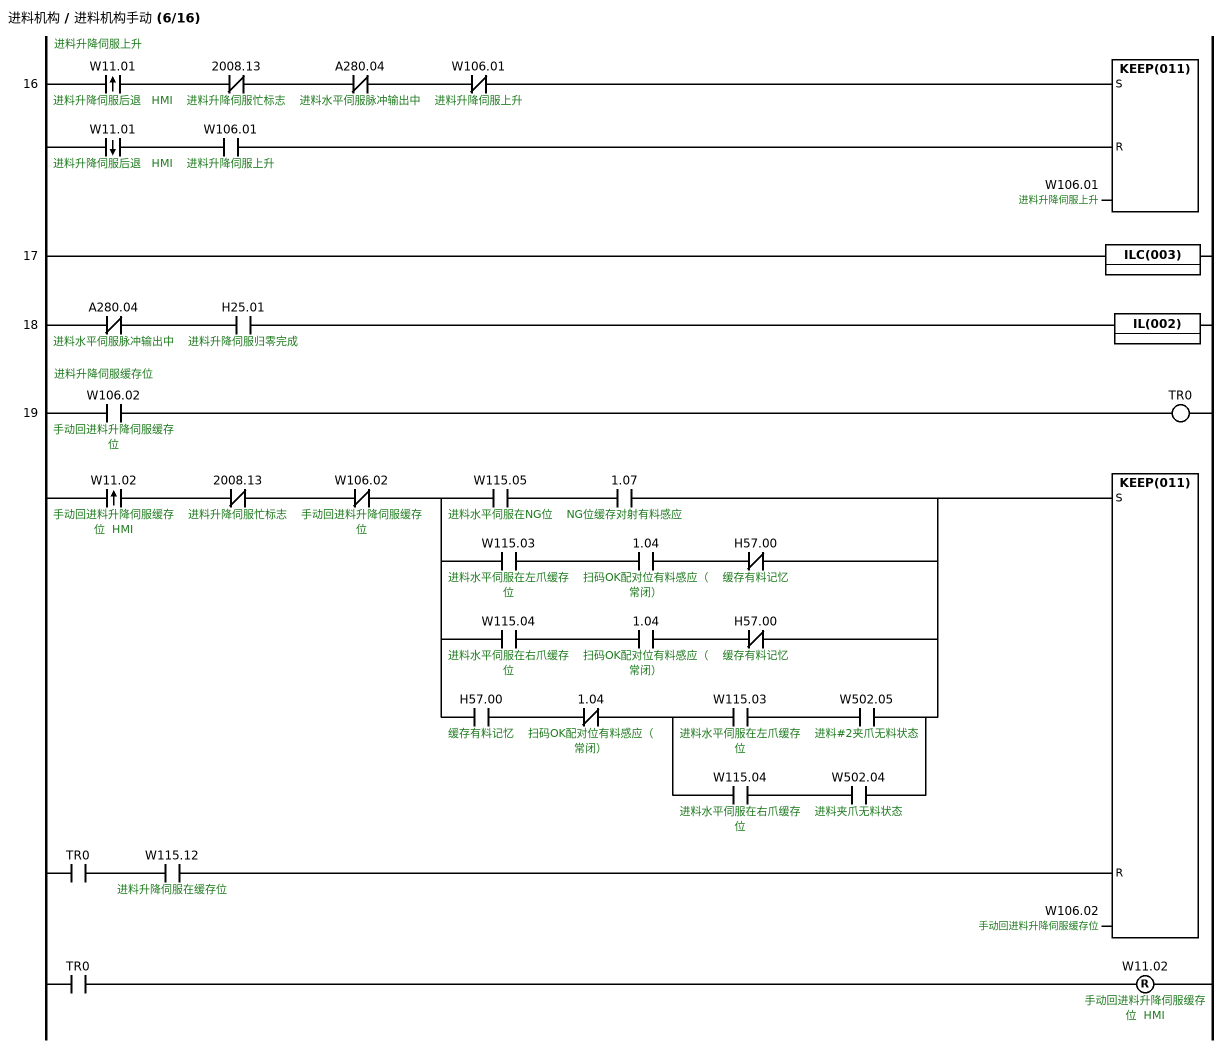
; [picture p120: 进料机构 / 进料机构手动, rungs 16-19]
; rung 16: 进料升降伺服上升
@LD W11.01  ; 进料升降伺服后退   HMI
ANDNOT 2008.13  ; 进料升降伺服忙标志
ANDNOT A280.04  ; 进料水平伺服脉冲输出中
ANDNOT W106.01  ; 进料升降伺服上升
%LD W11.01  ; 进料升降伺服后退   HMI
AND W106.01  ; 进料升降伺服上升
KEEP(011) W106.01  ; 进料升降伺服上升
; rung 17
ILC(003)
; rung 18
LDNOT A280.04  ; 进料水平伺服脉冲输出中
AND H25.01  ; 进料升降伺服归零完成
IL(002)
; rung 19: 进料升降伺服缓存位
@LD W11.02  ; 手动回进料升降伺服缓存位  HMI
ANDNOT 2008.13  ; 进料升降伺服忙标志
ANDNOT W106.02  ; 手动回进料升降伺服缓存位
LD W115.05  ; 进料水平伺服在NG位
AND 1.07  ; NG位缓存对射有料感应
LD W115.03  ; 进料水平伺服在左爪缓存位
AND 1.04  ; 扫码OK配对位有料感应（常闭）
ANDNOT H57.00  ; 缓存有料记忆
ORLD
LD W115.04  ; 进料水平伺服在右爪缓存位
AND 1.04  ; 扫码OK配对位有料感应（常闭）
ANDNOT H57.00  ; 缓存有料记忆
ORLD
LD H57.00  ; 缓存有料记忆
ANDNOT 1.04  ; 扫码OK配对位有料感应（常闭）
LD W115.03  ; 进料水平伺服在左爪缓存位
AND W502.05  ; 进料#2夹爪无料状态
LD W115.04  ; 进料水平伺服在右爪缓存位
AND W502.04  ; 进料夹爪无料状态
ORLD
ANDLD
ORLD
ANDLD
LD W106.02  ; 手动回进料升降伺服缓存位
OUT TR0
AND W115.12  ; 进料升降伺服在缓存位
KEEP(011) W106.02  ; 手动回进料升降伺服缓存位
LD TR0
RSET W11.02  ; 手动回进料升降伺服缓存位  HMI

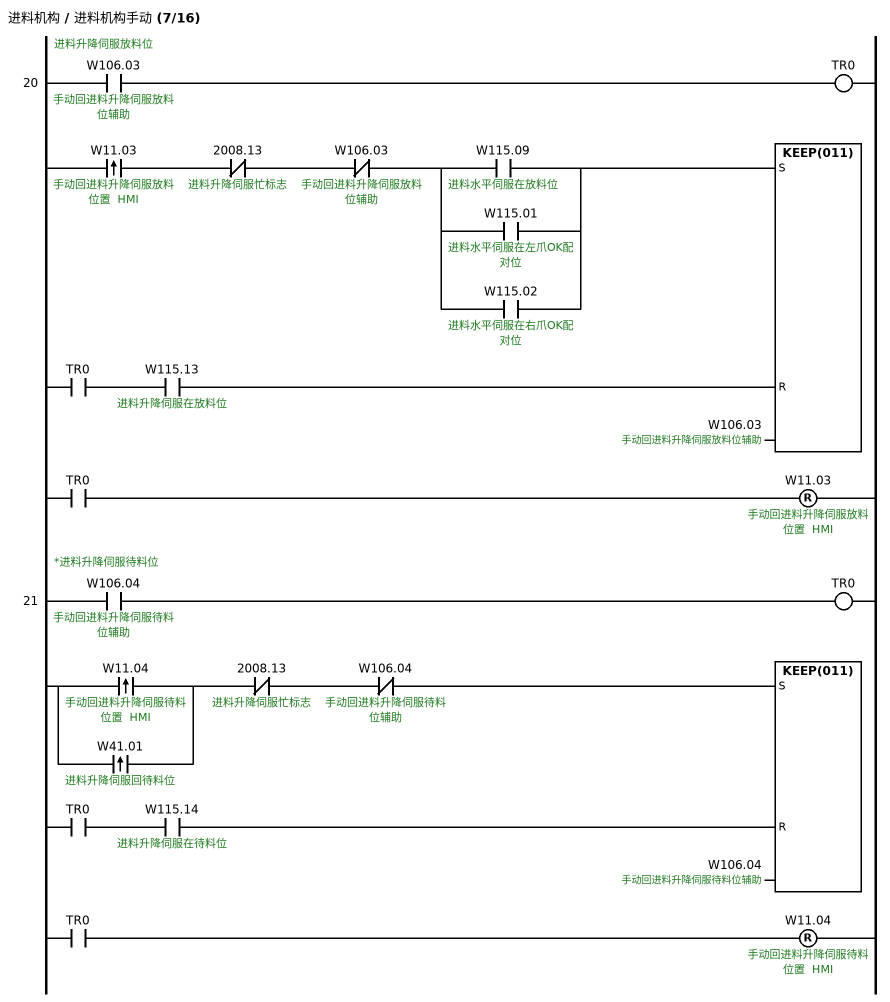
; rung 20: 进料升降伺服放料位
@LD W11.03  ; 手动回进料升降伺服放料位置  HMI
ANDNOT 2008.13  ; 进料升降伺服忙标志
ANDNOT W106.03  ; 手动回进料升降伺服放料位辅助
LD W115.09  ; 进料水平伺服在放料位
OR W115.01  ; 进料水平伺服在左爪OK配对位
OR W115.02  ; 进料水平伺服在右爪OK配对位
ANDLD
LD W106.03  ; 手动回进料升降伺服放料位辅助
OUT TR0
AND W115.13  ; 进料升降伺服在放料位
KEEP(011) W106.03  ; 手动回进料升降伺服放料位辅助
LD TR0
RSET W11.03  ; 手动回进料升降伺服放料位置  HMI
; rung 21: *进料升降伺服待料位
@LD W11.04  ; 手动回进料升降伺服待料位置  HMI
@OR W41.01  ; 进料升降伺服回待料位
ANDNOT 2008.13  ; 进料升降伺服忙标志
ANDNOT W106.04  ; 手动回进料升降伺服待料位辅助
LD W106.04  ; 手动回进料升降伺服待料位辅助
OUT TR0
AND W115.14  ; 进料升降伺服在待料位
KEEP(011) W106.04  ; 手动回进料升降伺服待料位辅助
LD TR0
RSET W11.04  ; 手动回进料升降伺服待料位置  HMI

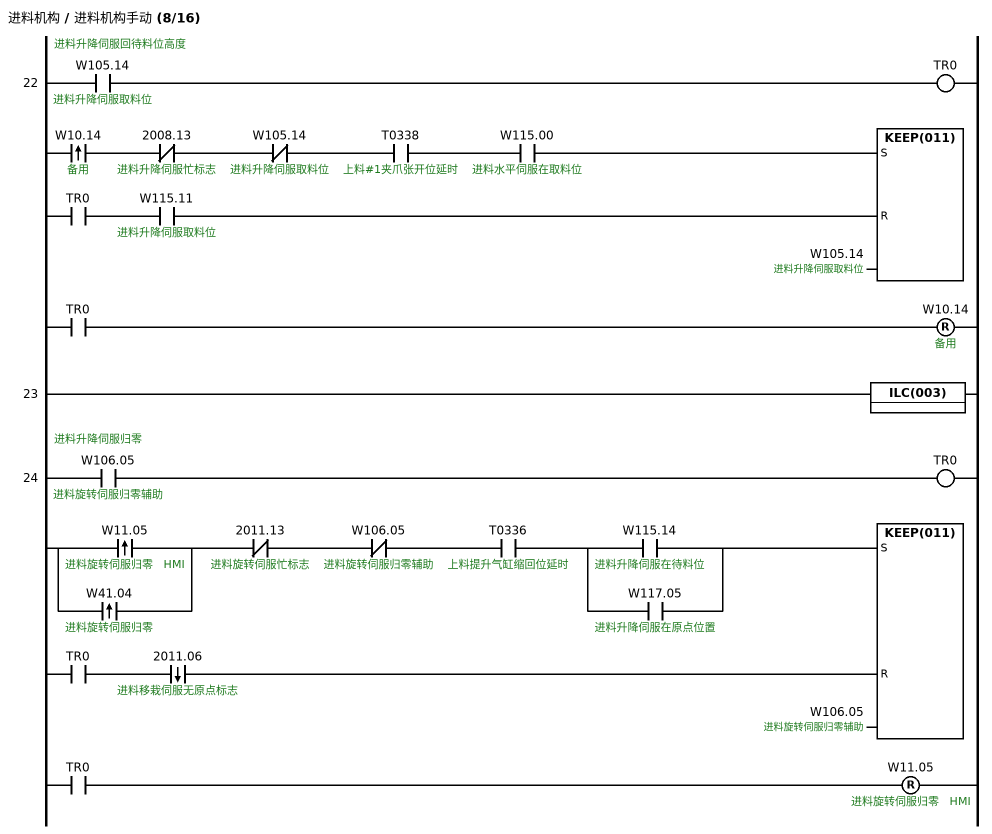
; rung 22: 进料升降伺服回待料位高度
@LD W10.14  ; 备用
ANDNOT 2008.13  ; 进料升降伺服忙标志
ANDNOT W105.14  ; 进料升降伺服取料位
AND T0338  ; 上料#1夹爪张开位延时
AND W115.00  ; 进料水平伺服在取料位
LD W105.14  ; 进料升降伺服取料位
OUT TR0
AND W115.11  ; 进料升降伺服取料位
KEEP(011) W105.14  ; 进料升降伺服取料位
LD TR0
RSET W10.14  ; 备用
; rung 23
ILC(003)
; rung 24: 进料升降伺服归零
@LD W11.05  ; 进料旋转伺服归零   HMI
@OR W41.04  ; 进料旋转伺服归零
ANDNOT 2011.13  ; 进料旋转伺服忙标志
ANDNOT W106.05  ; 进料旋转伺服归零辅助
AND T0336  ; 上料提升气缸缩回位延时
LD W115.14  ; 进料升降伺服在待料位
OR W117.05  ; 进料升降伺服在原点位置
ANDLD
LD W106.05  ; 进料旋转伺服归零辅助
OUT TR0
%AND 2011.06  ; 进料移栽伺服无原点标志
KEEP(011) W106.05  ; 进料旋转伺服归零辅助
LD TR0
RSET W11.05  ; 进料旋转伺服归零   HMI

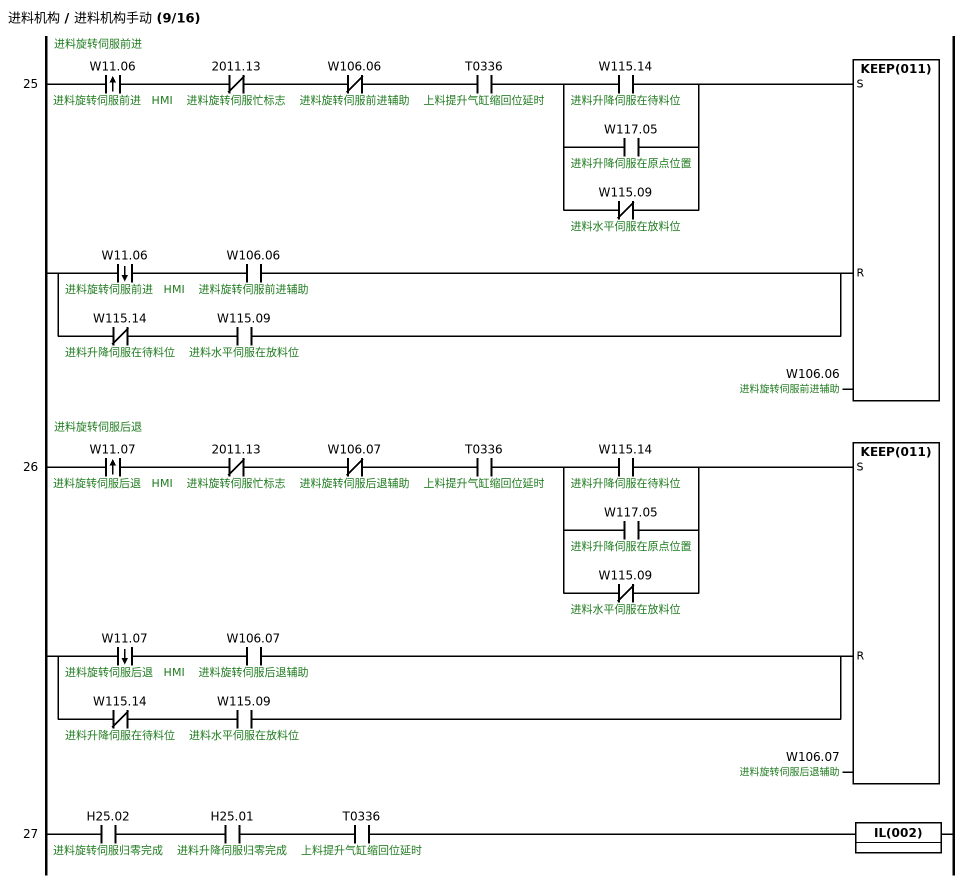
; rung 25: 进料旋转伺服前进
@LD W11.06  ; 进料旋转伺服前进   HMI
ANDNOT 2011.13  ; 进料旋转伺服忙标志
ANDNOT W106.06  ; 进料旋转伺服前进辅助
AND T0336  ; 上料提升气缸缩回位延时
LD W115.14  ; 进料升降伺服在待料位
OR W117.05  ; 进料升降伺服在原点位置
ORNOT W115.09  ; 进料水平伺服在放料位
ANDLD
%LD W11.06  ; 进料旋转伺服前进   HMI
AND W106.06  ; 进料旋转伺服前进辅助
LDNOT W115.14  ; 进料升降伺服在待料位
AND W115.09  ; 进料水平伺服在放料位
ORLD
KEEP(011) W106.06  ; 进料旋转伺服前进辅助
; rung 26: 进料旋转伺服后退
@LD W11.07  ; 进料旋转伺服后退   HMI
ANDNOT 2011.13  ; 进料旋转伺服忙标志
ANDNOT W106.07  ; 进料旋转伺服后退辅助
AND T0336  ; 上料提升气缸缩回位延时
LD W115.14  ; 进料升降伺服在待料位
OR W117.05  ; 进料升降伺服在原点位置
ORNOT W115.09  ; 进料水平伺服在放料位
ANDLD
%LD W11.07  ; 进料旋转伺服后退   HMI
AND W106.07  ; 进料旋转伺服后退辅助
LDNOT W115.14  ; 进料升降伺服在待料位
AND W115.09  ; 进料水平伺服在放料位
ORLD
KEEP(011) W106.07  ; 进料旋转伺服后退辅助
; rung 27
LD H25.02  ; 进料旋转伺服归零完成
AND H25.01  ; 进料升降伺服归零完成
AND T0336  ; 上料提升气缸缩回位延时
IL(002)

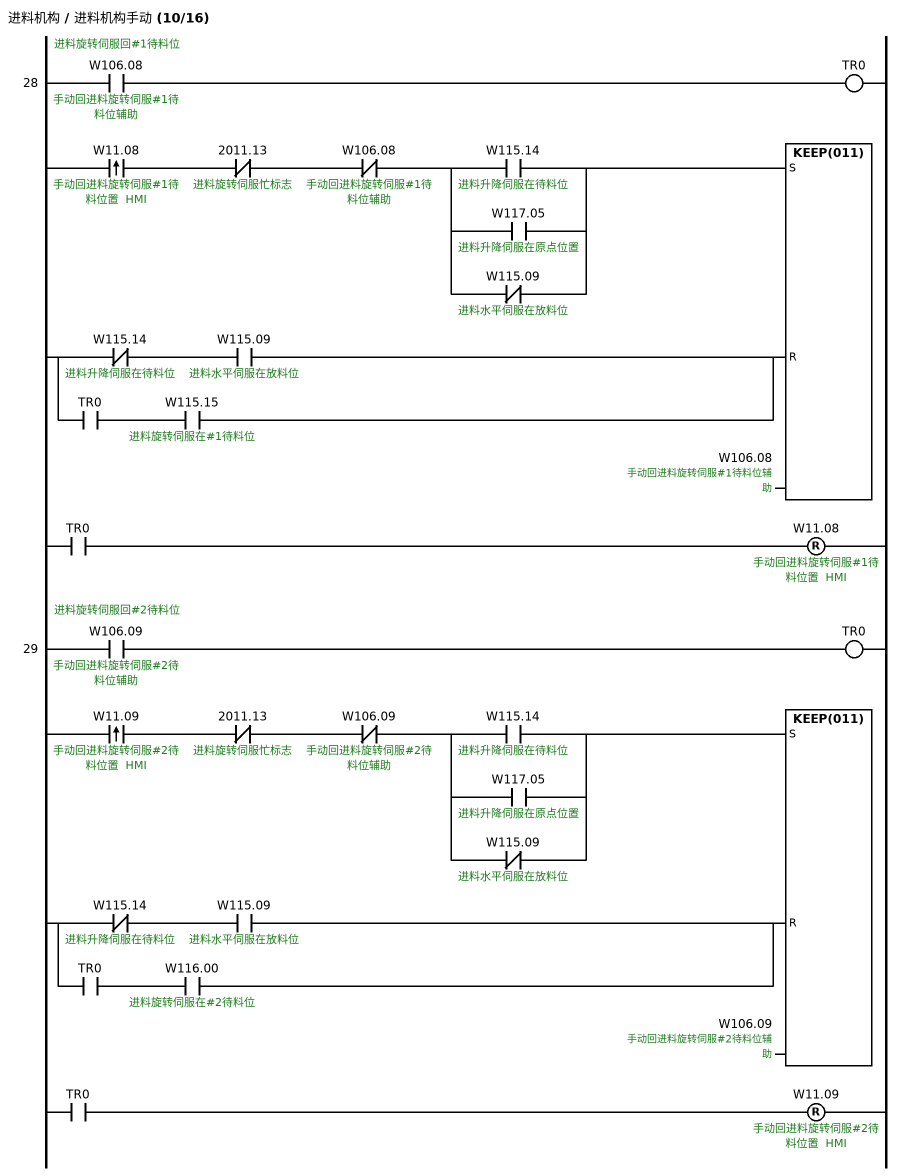
; rung 28: 进料旋转伺服回#1待料位
@LD W11.08  ; 手动回进料旋转伺服#1待料位置  HMI
ANDNOT 2011.13  ; 进料旋转伺服忙标志
ANDNOT W106.08  ; 手动回进料旋转伺服#1待料位辅助
LD W115.14  ; 进料升降伺服在待料位
OR W117.05  ; 进料升降伺服在原点位置
ORNOT W115.09  ; 进料水平伺服在放料位
ANDLD
LDNOT W115.14  ; 进料升降伺服在待料位
AND W115.09  ; 进料水平伺服在放料位
LD W106.08  ; 手动回进料旋转伺服#1待料位辅助
OUT TR0
AND W115.15  ; 进料旋转伺服在#1待料位
ORLD
KEEP(011) W106.08  ; 手动回进料旋转伺服#1待料位辅助
LD TR0
RSET W11.08  ; 手动回进料旋转伺服#1待料位置  HMI
; rung 29: 进料旋转伺服回#2待料位
@LD W11.09  ; 手动回进料旋转伺服#2待料位置  HMI
ANDNOT 2011.13  ; 进料旋转伺服忙标志
ANDNOT W106.09  ; 手动回进料旋转伺服#2待料位辅助
LD W115.14  ; 进料升降伺服在待料位
OR W117.05  ; 进料升降伺服在原点位置
ORNOT W115.09  ; 进料水平伺服在放料位
ANDLD
LDNOT W115.14  ; 进料升降伺服在待料位
AND W115.09  ; 进料水平伺服在放料位
LD W106.09  ; 手动回进料旋转伺服#2待料位辅助
OUT TR0
AND W116.00  ; 进料旋转伺服在#2待料位
ORLD
KEEP(011) W106.09  ; 手动回进料旋转伺服#2待料位辅助
LD TR0
RSET W11.09  ; 手动回进料旋转伺服#2待料位置  HMI

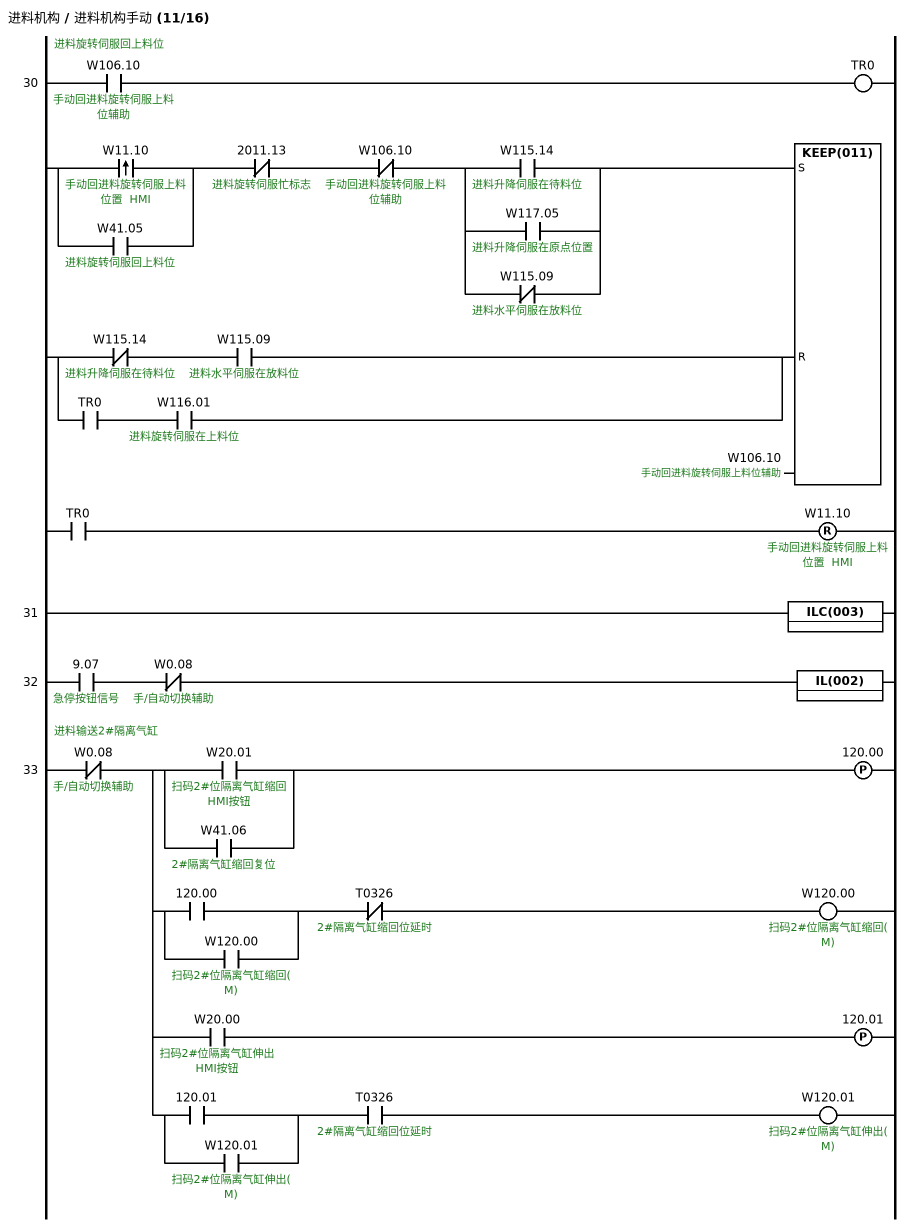
; rung 30: 进料旋转伺服回上料位
@LD W11.10  ; 手动回进料旋转伺服上料位置  HMI
OR W41.05  ; 进料旋转伺服回上料位
ANDNOT 2011.13  ; 进料旋转伺服忙标志
ANDNOT W106.10  ; 手动回进料旋转伺服上料位辅助
LD W115.14  ; 进料升降伺服在待料位
OR W117.05  ; 进料升降伺服在原点位置
ORNOT W115.09  ; 进料水平伺服在放料位
ANDLD
LDNOT W115.14  ; 进料升降伺服在待料位
AND W115.09  ; 进料水平伺服在放料位
LD W106.10  ; 手动回进料旋转伺服上料位辅助
OUT TR0
AND W116.01  ; 进料旋转伺服在上料位
ORLD
KEEP(011) W106.10  ; 手动回进料旋转伺服上料位辅助
LD TR0
RSET W11.10  ; 手动回进料旋转伺服上料位置  HMI
; rung 31
ILC(003)
; rung 32
LD 9.07  ; 急停按钮信号
ANDNOT W0.08  ; 手/自动切换辅助
IL(002)
; rung 33: 进料输送2#隔离气缸
LDNOT W0.08  ; 手/自动切换辅助
OUT TR0
LD W20.01  ; 扫码2#位隔离气缸缩回   HMI按钮
OR W41.06  ; 2#隔离气缸缩回复位
ANDLD
DIFU(013) 120.00
LD TR0
LD 120.00
OR W120.00  ; 扫码2#位隔离气缸缩回(M)
ANDLD
ANDNOT T0326  ; 2#隔离气缸缩回位延时
OUT W120.00  ; 扫码2#位隔离气缸缩回(M)
LD TR0
AND W20.00  ; 扫码2#位隔离气缸伸出   HMI按钮
DIFU(013) 120.01
LD TR0
LD 120.01
OR W120.01  ; 扫码2#位隔离气缸伸出(M)
ANDLD
AND T0326  ; 2#隔离气缸缩回位延时
OUT W120.01  ; 扫码2#位隔离气缸伸出(M)

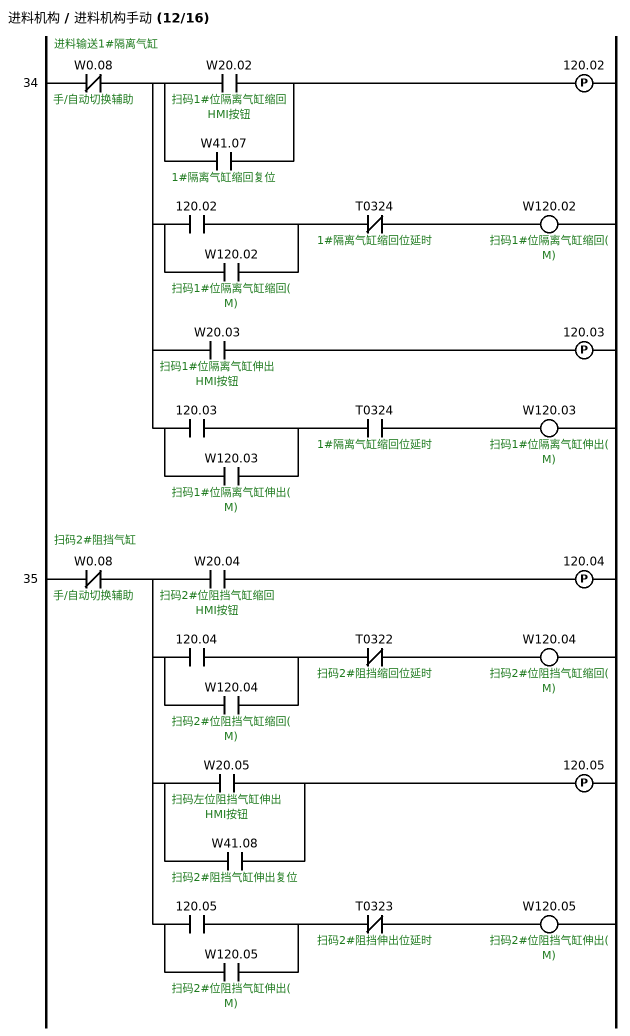
; rung 34: 进料输送1#隔离气缸
LDNOT W0.08  ; 手/自动切换辅助
OUT TR0
LD W20.02  ; 扫码1#位隔离气缸缩回   HMI按钮
OR W41.07  ; 1#隔离气缸缩回复位
ANDLD
DIFU(013) 120.02
LD TR0
LD 120.02
OR W120.02  ; 扫码1#位隔离气缸缩回(M)
ANDLD
ANDNOT T0324  ; 1#隔离气缸缩回位延时
OUT W120.02  ; 扫码1#位隔离气缸缩回(M)
LD TR0
AND W20.03  ; 扫码1#位隔离气缸伸出   HMI按钮
DIFU(013) 120.03
LD TR0
LD 120.03
OR W120.03  ; 扫码1#位隔离气缸伸出(M)
ANDLD
AND T0324  ; 1#隔离气缸缩回位延时
OUT W120.03  ; 扫码1#位隔离气缸伸出(M)
; rung 35: 扫码2#阻挡气缸
LDNOT W0.08  ; 手/自动切换辅助
OUT TR0
AND W20.04  ; 扫码2#位阻挡气缸缩回   HMI按钮
DIFU(013) 120.04
LD TR0
LD 120.04
OR W120.04  ; 扫码2#位阻挡气缸缩回(M)
ANDLD
ANDNOT T0322  ; 扫码2#阻挡缩回位延时
OUT W120.04  ; 扫码2#位阻挡气缸缩回(M)
LD TR0
LD W20.05  ; 扫码左位阻挡气缸伸出  HMI按钮
OR W41.08  ; 扫码2#阻挡气缸伸出复位
ANDLD
DIFU(013) 120.05
LD TR0
LD 120.05
OR W120.05  ; 扫码2#位阻挡气缸伸出(M)
ANDLD
ANDNOT T0323  ; 扫码2#阻挡伸出位延时
OUT W120.05  ; 扫码2#位阻挡气缸伸出(M)

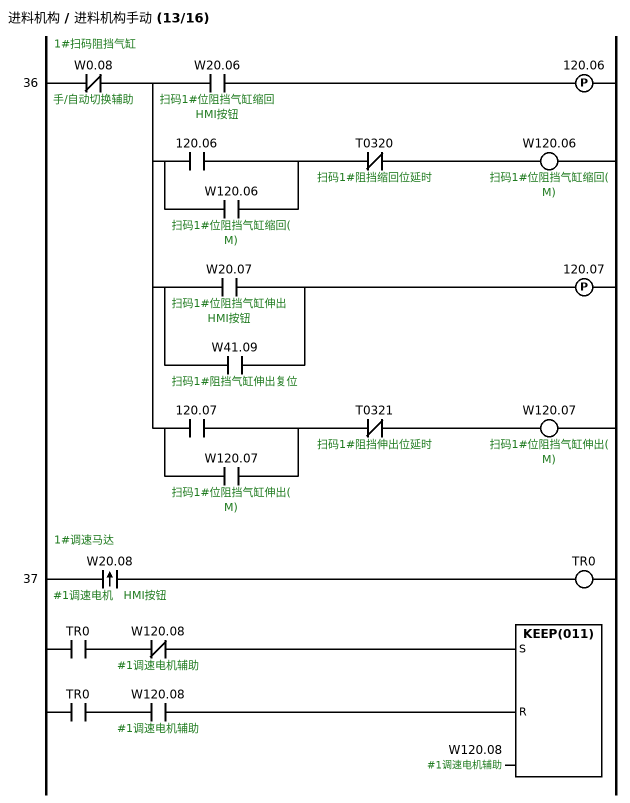
; rung 36: 1#扫码阻挡气缸
LDNOT W0.08  ; 手/自动切换辅助
OUT TR0
AND W20.06  ; 扫码1#位阻挡气缸缩回   HMI按钮
DIFU(013) 120.06
LD TR0
LD 120.06
OR W120.06  ; 扫码1#位阻挡气缸缩回(M)
ANDLD
ANDNOT T0320  ; 扫码1#阻挡缩回位延时
OUT W120.06  ; 扫码1#位阻挡气缸缩回(M)
LD TR0
LD W20.07  ; 扫码1#位阻挡气缸伸出   HMI按钮
OR W41.09  ; 扫码1#阻挡气缸伸出复位
ANDLD
DIFU(013) 120.07
LD TR0
LD 120.07
OR W120.07  ; 扫码1#位阻挡气缸伸出(M)
ANDLD
ANDNOT T0321  ; 扫码1#阻挡伸出位延时
OUT W120.07  ; 扫码1#位阻挡气缸伸出(M)
; rung 37: 1#调速马达
@LD W20.08  ; #1调速电机   HMI按钮
OUT TR0
ANDNOT W120.08  ; #1调速电机辅助
LD TR0
AND W120.08  ; #1调速电机辅助
KEEP(011) W120.08  ; #1调速电机辅助

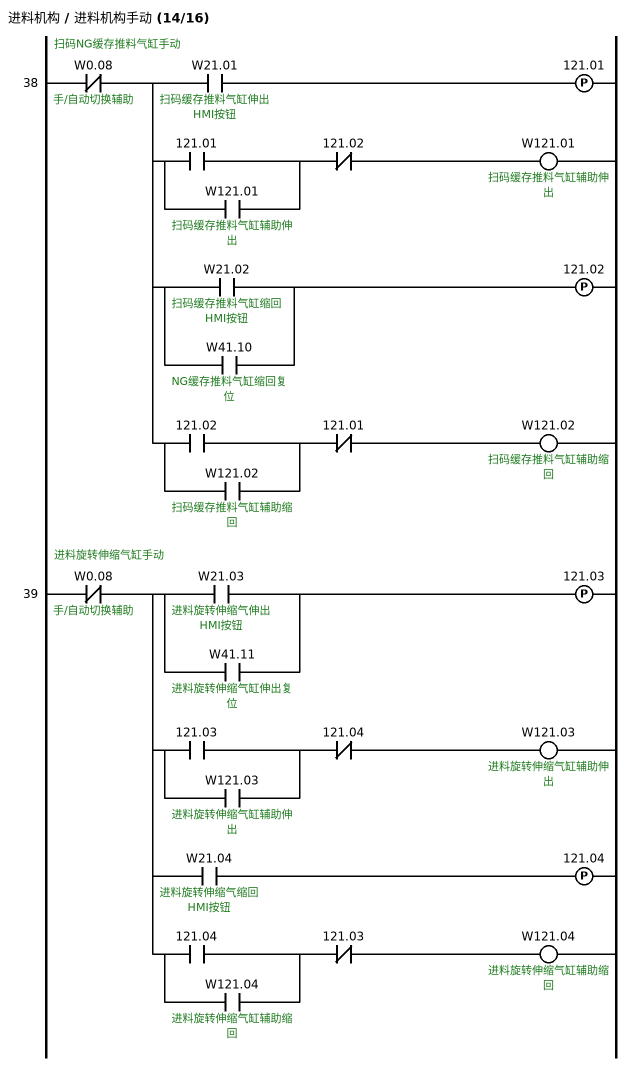
; rung 38: 扫码NG缓存推料气缸手动
LDNOT W0.08  ; 手/自动切换辅助
OUT TR0
AND W21.01  ; 扫码缓存推料气缸伸出   HMI按钮
DIFU(013) 121.01
LD TR0
LD 121.01
OR W121.01  ; 扫码缓存推料气缸辅助伸出
ANDLD
ANDNOT 121.02
OUT W121.01  ; 扫码缓存推料气缸辅助伸出
LD TR0
LD W21.02  ; 扫码缓存推料气缸缩回   HMI按钮
OR W41.10  ; NG缓存推料气缸缩回复位
ANDLD
DIFU(013) 121.02
LD TR0
LD 121.02
OR W121.02  ; 扫码缓存推料气缸辅助缩回
ANDLD
ANDNOT 121.01
OUT W121.02  ; 扫码缓存推料气缸辅助缩回
; rung 39: 进料旋转伸缩气缸手动
LDNOT W0.08  ; 手/自动切换辅助
OUT TR0
LD W21.03  ; 进料旋转伸缩气伸出   HMI按钮
OR W41.11  ; 进料旋转伸缩气缸伸出复位
ANDLD
DIFU(013) 121.03
LD TR0
LD 121.03
OR W121.03  ; 进料旋转伸缩气缸辅助伸出
ANDLD
ANDNOT 121.04
OUT W121.03  ; 进料旋转伸缩气缸辅助伸出
LD TR0
AND W21.04  ; 进料旋转伸缩气缩回   HMI按钮
DIFU(013) 121.04
LD TR0
LD 121.04
OR W121.04  ; 进料旋转伸缩气缸辅助缩回
ANDLD
ANDNOT 121.03
OUT W121.04  ; 进料旋转伸缩气缸辅助缩回

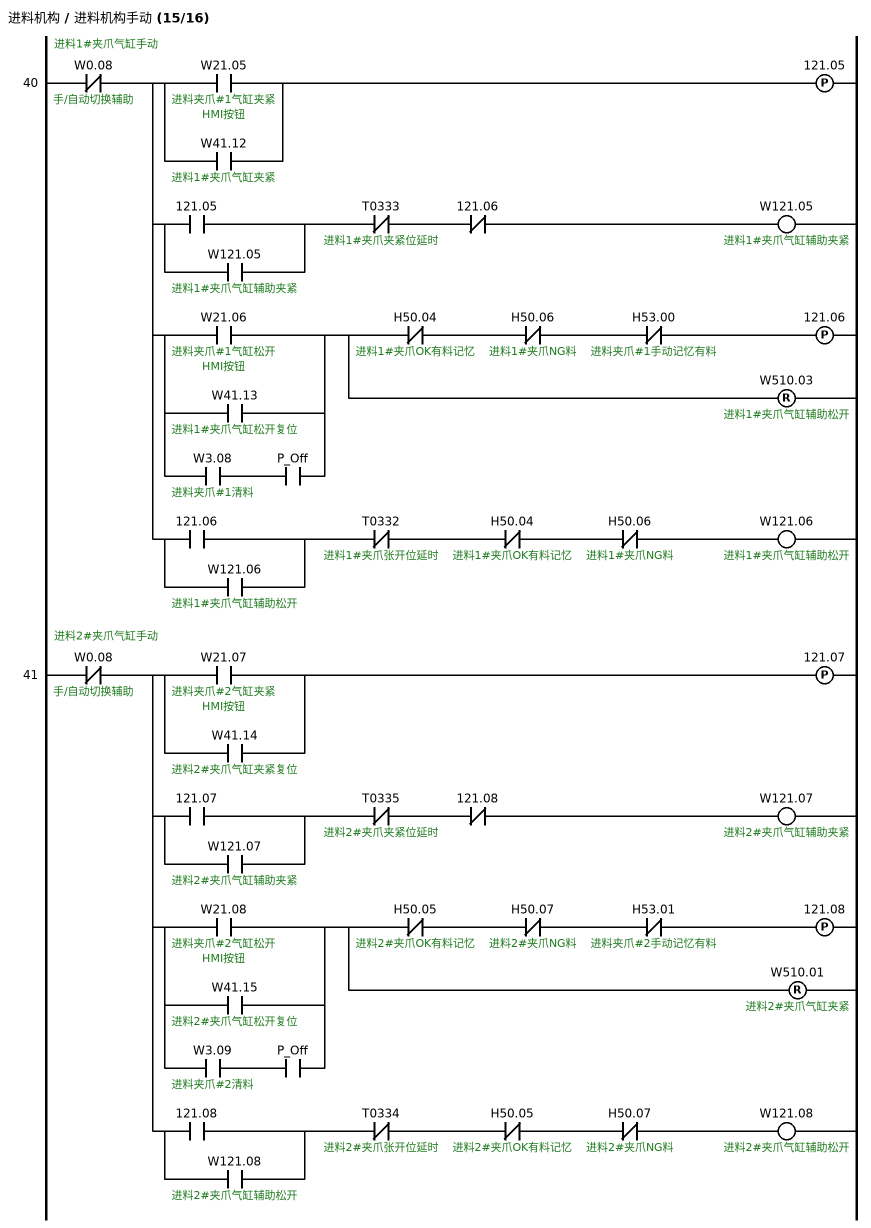
; rung 40: 进料1#夹爪气缸手动
LDNOT W0.08  ; 手/自动切换辅助
OUT TR0
LD W21.05  ; 进料夹爪#1气缸夹紧   HMI按钮
OR W41.12  ; 进料1#夹爪气缸夹紧
ANDLD
DIFU(013) 121.05
LD TR0
LD 121.05
OR W121.05  ; 进料1#夹爪气缸辅助夹紧
ANDLD
ANDNOT T0333  ; 进料1#夹爪夹紧位延时
ANDNOT 121.06
OUT W121.05  ; 进料1#夹爪气缸辅助夹紧
LD TR0
LD W21.06  ; 进料夹爪#1气缸松开   HMI按钮
OR W41.13  ; 进料1#夹爪气缸松开复位
LD W3.08  ; 进料夹爪#1清料
AND P_Off
ORLD
ANDLD
OUT TR1
ANDNOT H50.04  ; 进料1#夹爪OK有料记忆
ANDNOT H50.06  ; 进料1#夹爪NG料
ANDNOT H53.00  ; 进料夹爪#1手动记忆有料
DIFU(013) 121.06
LD TR1
RSET W510.03  ; 进料1#夹爪气缸辅助松开
LD TR0
LD 121.06
OR W121.06  ; 进料1#夹爪气缸辅助松开
ANDLD
ANDNOT T0332  ; 进料1#夹爪张开位延时
ANDNOT H50.04  ; 进料1#夹爪OK有料记忆
ANDNOT H50.06  ; 进料1#夹爪NG料
OUT W121.06  ; 进料1#夹爪气缸辅助松开
; rung 41: 进料2#夹爪气缸手动
LDNOT W0.08  ; 手/自动切换辅助
OUT TR0
LD W21.07  ; 进料夹爪#2气缸夹紧   HMI按钮
OR W41.14  ; 进料2#夹爪气缸夹紧复位
ANDLD
DIFU(013) 121.07
LD TR0
LD 121.07
OR W121.07  ; 进料2#夹爪气缸辅助夹紧
ANDLD
ANDNOT T0335  ; 进料2#夹爪夹紧位延时
ANDNOT 121.08
OUT W121.07  ; 进料2#夹爪气缸辅助夹紧
LD TR0
LD W21.08  ; 进料夹爪#2气缸松开   HMI按钮
OR W41.15  ; 进料2#夹爪气缸松开复位
LD W3.09  ; 进料夹爪#2清料
AND P_Off
ORLD
ANDLD
OUT TR1
ANDNOT H50.05  ; 进料2#夹爪OK有料记忆
ANDNOT H50.07  ; 进料2#夹爪NG料
ANDNOT H53.01  ; 进料夹爪#2手动记忆有料
DIFU(013) 121.08
LD TR1
RSET W510.01  ; 进料2#夹爪气缸夹紧
LD TR0
LD 121.08
OR W121.08  ; 进料2#夹爪气缸辅助松开
ANDLD
ANDNOT T0334  ; 进料2#夹爪张开位延时
ANDNOT H50.05  ; 进料2#夹爪OK有料记忆
ANDNOT H50.07  ; 进料2#夹爪NG料
OUT W121.08  ; 进料2#夹爪气缸辅助松开

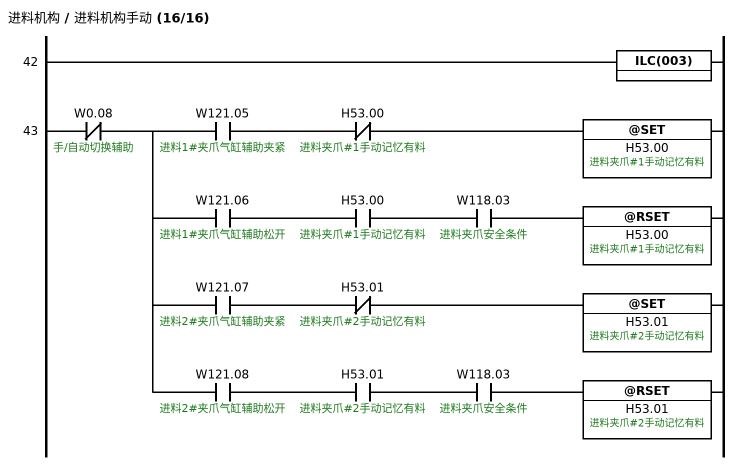
; rung 42
ILC(003)
; rung 43
LDNOT W0.08  ; 手/自动切换辅助
OUT TR0
AND W121.05  ; 进料1#夹爪气缸辅助夹紧
ANDNOT H53.00  ; 进料夹爪#1手动记忆有料
@SET H53.00  ; 进料夹爪#1手动记忆有料
LD TR0
AND W121.06  ; 进料1#夹爪气缸辅助松开
AND H53.00  ; 进料夹爪#1手动记忆有料
AND W118.03  ; 进料夹爪安全条件
@RSET H53.00  ; 进料夹爪#1手动记忆有料
LD TR0
AND W121.07  ; 进料2#夹爪气缸辅助夹紧
ANDNOT H53.01  ; 进料夹爪#2手动记忆有料
@SET H53.01  ; 进料夹爪#2手动记忆有料
LD TR0
AND W121.08  ; 进料2#夹爪气缸辅助松开
AND H53.01  ; 进料夹爪#2手动记忆有料
AND W118.03  ; 进料夹爪安全条件
@RSET H53.01  ; 进料夹爪#2手动记忆有料

### Section 进料水平伺服参数设置

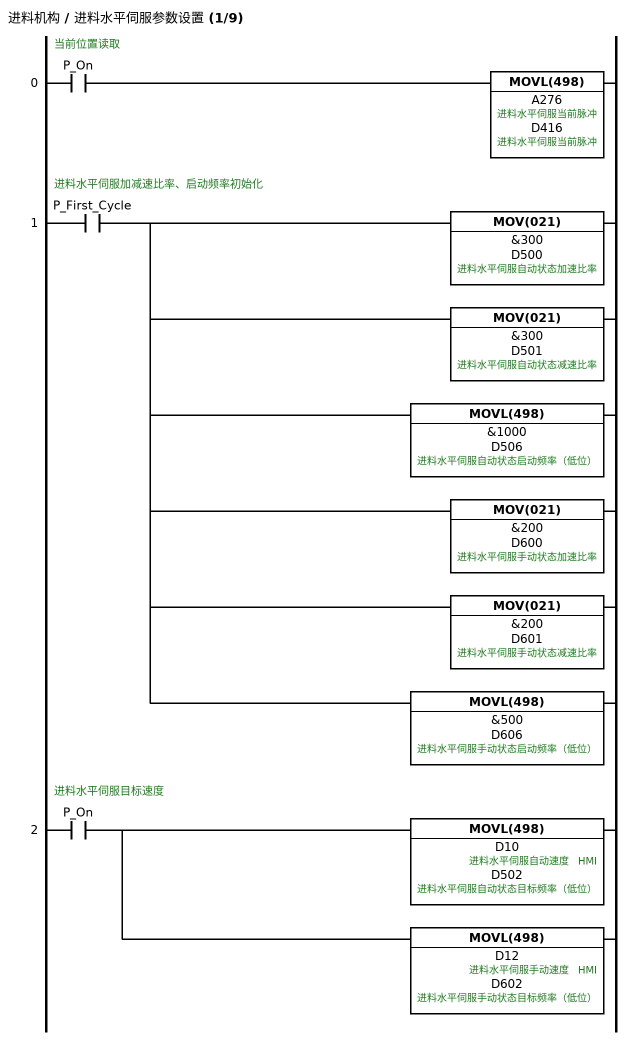
; rung 0: 当前位置读取
LD P_On
MOVL(498) A276 D416  ; 进料水平伺服当前脉冲
; rung 1: 进料水平伺服加减速比率、启动频率初始化
LD P_First_Cycle
MOV(021) &300 D500  ; 进料水平伺服自动状态加速比率
MOV(021) &300 D501  ; 进料水平伺服自动状态减速比率
MOVL(498) &1000 D506  ; 进料水平伺服自动状态启动频率（低位）
MOV(021) &200 D600  ; 进料水平伺服手动状态加速比率
MOV(021) &200 D601  ; 进料水平伺服手动状态减速比率
MOVL(498) &500 D606  ; 进料水平伺服手动状态启动频率（低位）
; rung 2: 进料水平伺服目标速度
LD P_On
MOVL(498) D10 D502  ; 进料水平伺服自动速度   HMI, 进料水平伺服自动状态目标频率（低位）
MOVL(498) D12 D602  ; 进料水平伺服手动速度   HMI, 进料水平伺服手动状态目标频率（低位）

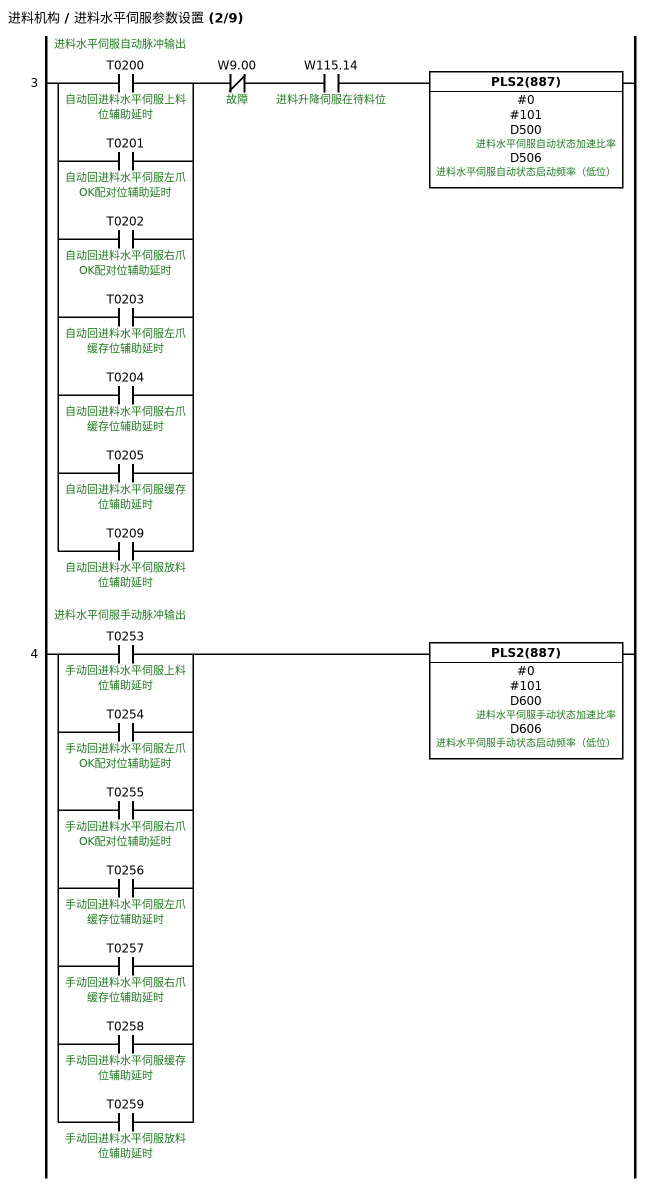
; rung 3: 进料水平伺服自动脉冲输出
LD T0200  ; 自动回进料水平伺服上料位辅助延时
OR T0201  ; 自动回进料水平伺服左爪OK配对位辅助延时
OR T0202  ; 自动回进料水平伺服右爪OK配对位辅助延时
OR T0203  ; 自动回进料水平伺服左爪缓存位辅助延时
OR T0204  ; 自动回进料水平伺服右爪缓存位辅助延时
OR T0205  ; 自动回进料水平伺服缓存位辅助延时
OR T0209  ; 自动回进料水平伺服放料位辅助延时
ANDNOT W9.00  ; 故障
AND W115.14  ; 进料升降伺服在待料位
PLS2(887) #0 #101 D500 D506  ; 进料水平伺服自动状态加速比率, 进料水平伺服自动状态启动频率（低位）
; rung 4: 进料水平伺服手动脉冲输出
LD T0253  ; 手动回进料水平伺服上料位辅助延时
OR T0254  ; 手动回进料水平伺服左爪OK配对位辅助延时
OR T0255  ; 手动回进料水平伺服右爪OK配对位辅助延时
OR T0256  ; 手动回进料水平伺服左爪缓存位辅助延时
OR T0257  ; 手动回进料水平伺服右爪缓存位辅助延时
OR T0258  ; 手动回进料水平伺服缓存位辅助延时
OR T0259  ; 手动回进料水平伺服放料位辅助延时
PLS2(887) #0 #101 D600 D606  ; 进料水平伺服手动状态加速比率, 进料水平伺服手动状态启动频率（低位）

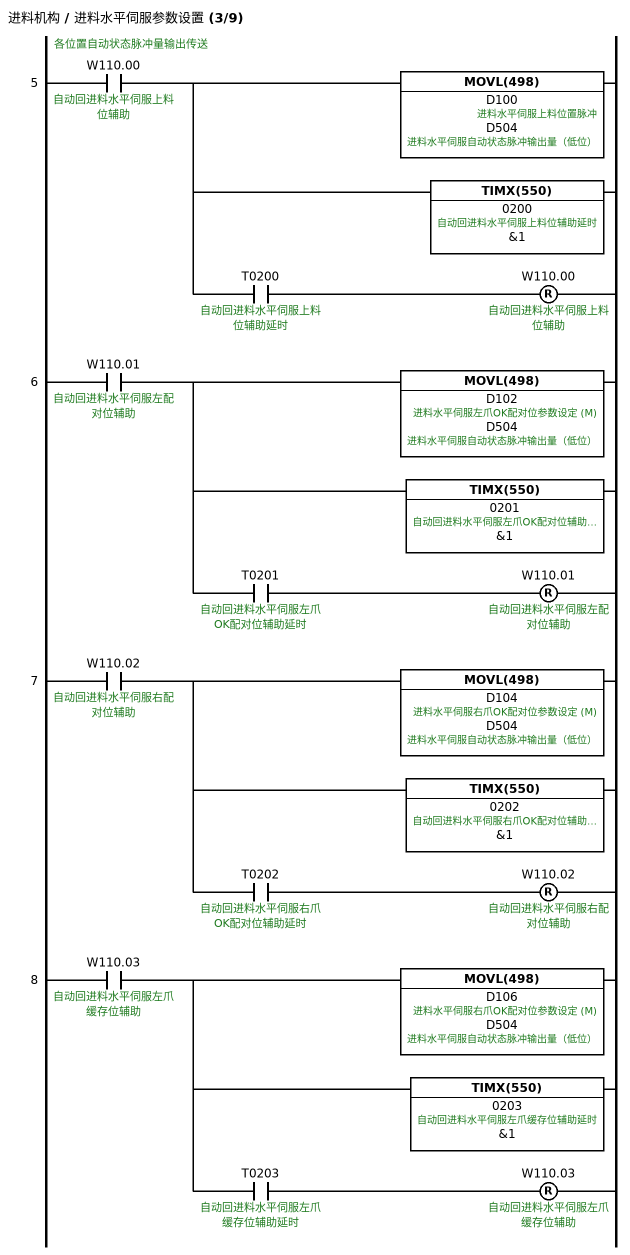
; rung 5: 各位置自动状态脉冲量输出传送
LD W110.00  ; 自动回进料水平伺服上料位辅助
MOVL(498) D100 D504  ; 进料水平伺服上料位置脉冲, 进料水平伺服自动状态脉冲输出量（低位）
TIMX(550) 0200 &1  ; 自动回进料水平伺服上料位辅助延时
AND T0200  ; 自动回进料水平伺服上料位辅助延时
RSET W110.00  ; 自动回进料水平伺服上料位辅助
; rung 6
LD W110.01  ; 自动回进料水平伺服左配对位辅助
MOVL(498) D102 D504  ; 进料水平伺服左爪OK配对位参数设定 (M), 进料水平伺服自动状态脉冲输出量（低位）
TIMX(550) 0201 &1  ; 自动回进料水平伺服左爪OK配对位辅助延时
AND T0201  ; 自动回进料水平伺服左爪OK配对位辅助延时
RSET W110.01  ; 自动回进料水平伺服左配对位辅助
; rung 7
LD W110.02  ; 自动回进料水平伺服右配对位辅助
MOVL(498) D104 D504  ; 进料水平伺服右爪OK配对位参数设定 (M), 进料水平伺服自动状态脉冲输出量（低位）
TIMX(550) 0202 &1  ; 自动回进料水平伺服右爪OK配对位辅助延时
AND T0202  ; 自动回进料水平伺服右爪OK配对位辅助延时
RSET W110.02  ; 自动回进料水平伺服右配对位辅助
; rung 8
LD W110.03  ; 自动回进料水平伺服左爪缓存位辅助
MOVL(498) D106 D504  ; 进料水平伺服右爪OK配对位参数设定 (M), 进料水平伺服自动状态脉冲输出量（低位）
TIMX(550) 0203 &1  ; 自动回进料水平伺服左爪缓存位辅助延时
AND T0203  ; 自动回进料水平伺服左爪缓存位辅助延时
RSET W110.03  ; 自动回进料水平伺服左爪缓存位辅助

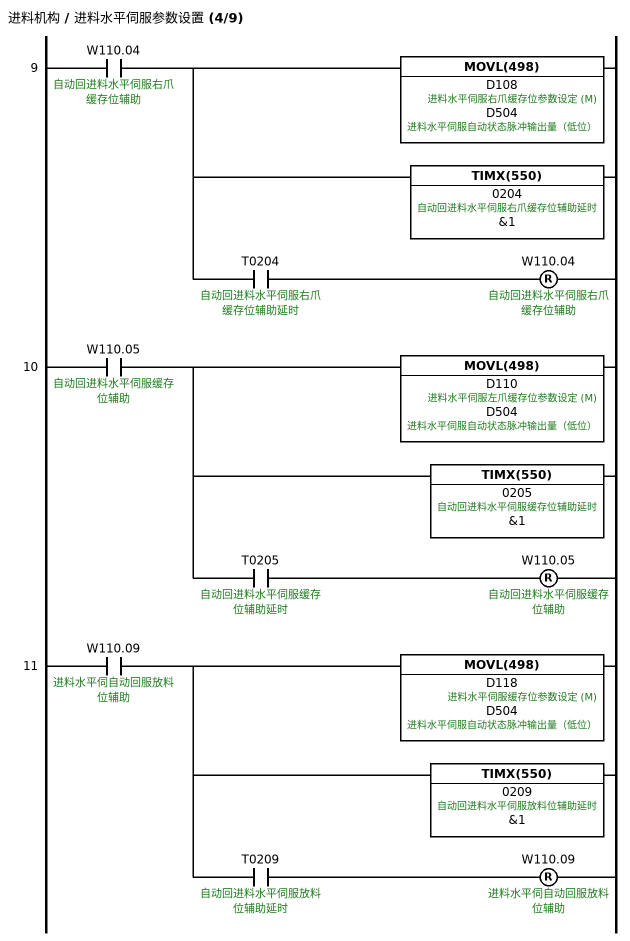
; rung 9
LD W110.04  ; 自动回进料水平伺服右爪缓存位辅助
MOVL(498) D108 D504  ; 进料水平伺服右爪缓存位参数设定 (M), 进料水平伺服自动状态脉冲输出量（低位）
TIMX(550) 0204 &1  ; 自动回进料水平伺服右爪缓存位辅助延时
AND T0204  ; 自动回进料水平伺服右爪缓存位辅助延时
RSET W110.04  ; 自动回进料水平伺服右爪缓存位辅助
; rung 10
LD W110.05  ; 自动回进料水平伺服缓存位辅助
MOVL(498) D110 D504  ; 进料水平伺服左爪缓存位参数设定 (M), 进料水平伺服自动状态脉冲输出量（低位）
TIMX(550) 0205 &1  ; 自动回进料水平伺服缓存位辅助延时
AND T0205  ; 自动回进料水平伺服缓存位辅助延时
RSET W110.05  ; 自动回进料水平伺服缓存位辅助
; rung 11
LD W110.09  ; 进料水平伺自动回服放料位辅助
MOVL(498) D118 D504  ; 进料水平伺服缓存位参数设定 (M), 进料水平伺服自动状态脉冲输出量（低位）
TIMX(550) 0209 &1  ; 自动回进料水平伺服放料位辅助延时
AND T0209  ; 自动回进料水平伺服放料位辅助延时
RSET W110.09  ; 进料水平伺自动回服放料位辅助

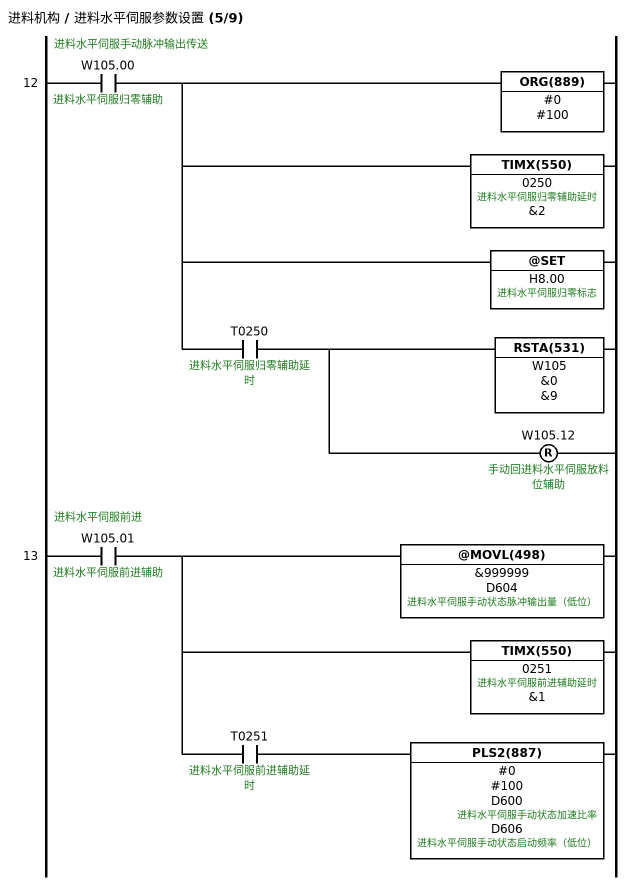
; rung 12: 进料水平伺服手动脉冲输出传送
LD W105.00  ; 进料水平伺服归零辅助
ORG(889) #0 #100
TIMX(550) 0250 &2  ; 进料水平伺服归零辅助延时
@SET H8.00  ; 进料水平伺服归零标志
AND T0250  ; 进料水平伺服归零辅助延时
RSTA(531) W105 &0 &9
RSET W105.12  ; 手动回进料水平伺服放料位辅助
; rung 13: 进料水平伺服前进
LD W105.01  ; 进料水平伺服前进辅助
@MOVL(498) &999999 D604  ; 进料水平伺服手动状态脉冲输出量（低位）
TIMX(550) 0251 &1  ; 进料水平伺服前进辅助延时
AND T0251  ; 进料水平伺服前进辅助延时
PLS2(887) #0 #100 D600 D606  ; 进料水平伺服手动状态加速比率, 进料水平伺服手动状态启动频率（低位）

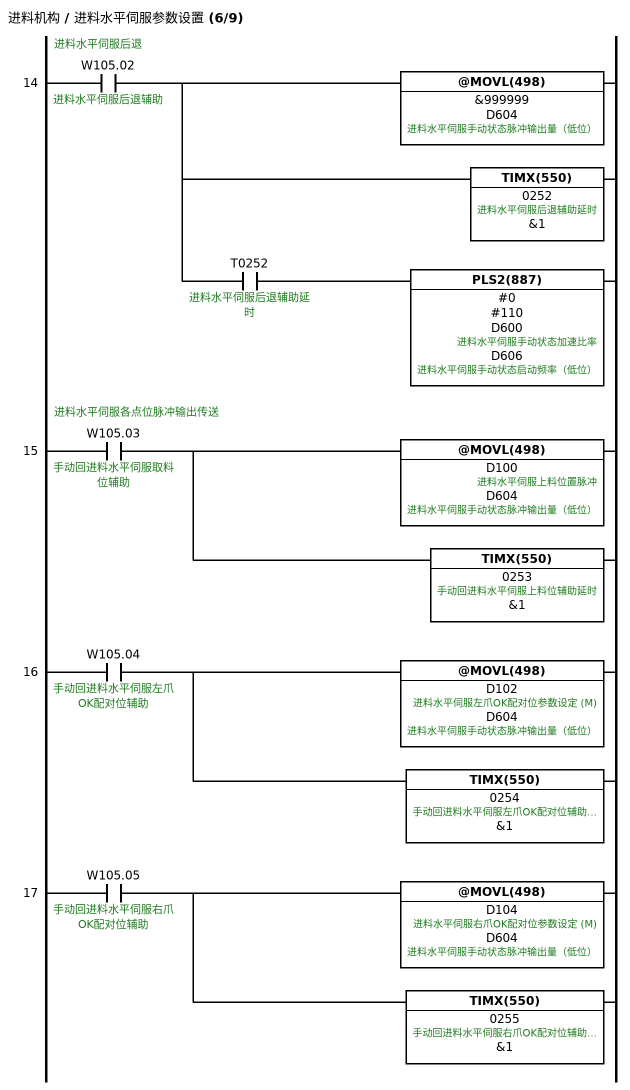
; rung 14: 进料水平伺服后退
LD W105.02  ; 进料水平伺服后退辅助
@MOVL(498) &999999 D604  ; 进料水平伺服手动状态脉冲输出量（低位）
TIMX(550) 0252 &1  ; 进料水平伺服后退辅助延时
AND T0252  ; 进料水平伺服后退辅助延时
PLS2(887) #0 #110 D600 D606  ; 进料水平伺服手动状态加速比率, 进料水平伺服手动状态启动频率（低位）
; rung 15: 进料水平伺服各点位脉冲输出传送
LD W105.03  ; 手动回进料水平伺服取料位辅助
@MOVL(498) D100 D604  ; 进料水平伺服上料位置脉冲, 进料水平伺服手动状态脉冲输出量（低位）
TIMX(550) 0253 &1  ; 手动回进料水平伺服上料位辅助延时
; rung 16
LD W105.04  ; 手动回进料水平伺服左爪OK配对位辅助
@MOVL(498) D102 D604  ; 进料水平伺服左爪OK配对位参数设定 (M), 进料水平伺服手动状态脉冲输出量（低位）
TIMX(550) 0254 &1  ; 手动回进料水平伺服左爪OK配对位辅助延时
; rung 17
LD W105.05  ; 手动回进料水平伺服右爪OK配对位辅助
@MOVL(498) D104 D604  ; 进料水平伺服右爪OK配对位参数设定 (M), 进料水平伺服手动状态脉冲输出量（低位）
TIMX(550) 0255 &1  ; 手动回进料水平伺服右爪OK配对位辅助延时

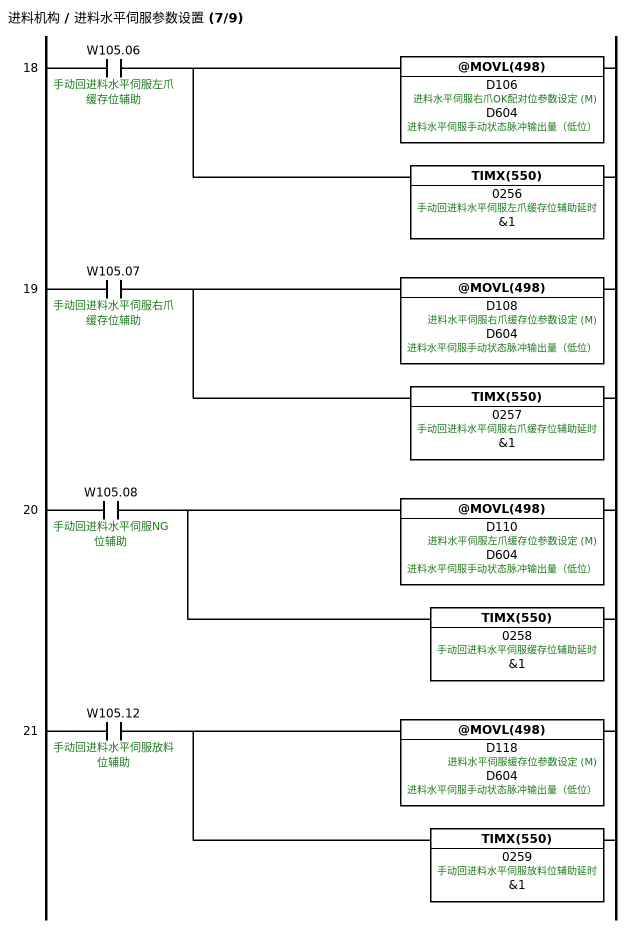
; rung 18
LD W105.06  ; 手动回进料水平伺服左爪缓存位辅助
@MOVL(498) D106 D604  ; 进料水平伺服右爪OK配对位参数设定 (M), 进料水平伺服手动状态脉冲输出量（低位）
TIMX(550) 0256 &1  ; 手动回进料水平伺服左爪缓存位辅助延时
; rung 19
LD W105.07  ; 手动回进料水平伺服右爪缓存位辅助
@MOVL(498) D108 D604  ; 进料水平伺服右爪缓存位参数设定 (M), 进料水平伺服手动状态脉冲输出量（低位）
TIMX(550) 0257 &1  ; 手动回进料水平伺服右爪缓存位辅助延时
; rung 20
LD W105.08  ; 手动回进料水平伺服NG位辅助
@MOVL(498) D110 D604  ; 进料水平伺服左爪缓存位参数设定 (M), 进料水平伺服手动状态脉冲输出量（低位）
TIMX(550) 0258 &1  ; 手动回进料水平伺服缓存位辅助延时
; rung 21
LD W105.12  ; 手动回进料水平伺服放料位辅助
@MOVL(498) D118 D604  ; 进料水平伺服缓存位参数设定 (M), 进料水平伺服手动状态脉冲输出量（低位）
TIMX(550) 0259 &1  ; 手动回进料水平伺服放料位辅助延时

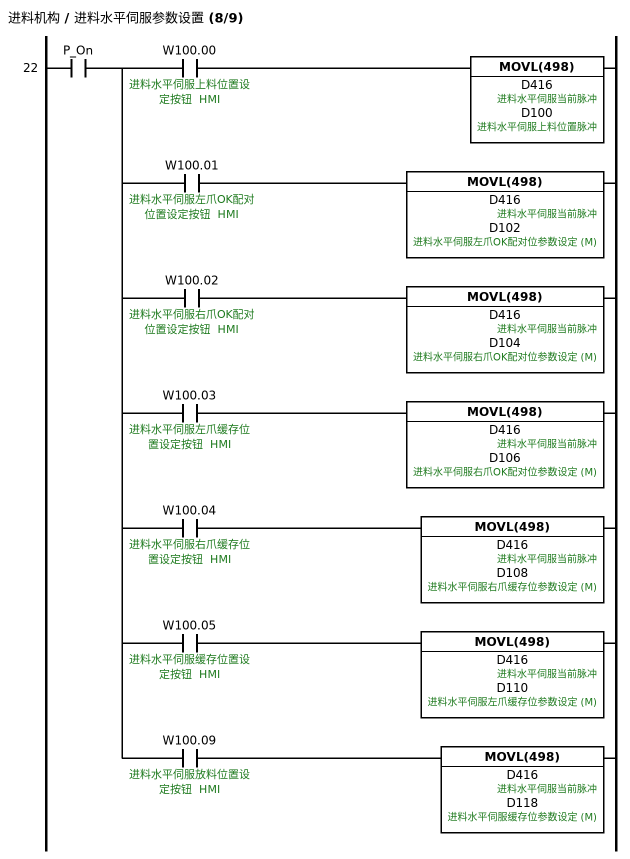
; rung 22
LD P_On
OUT TR0
AND W100.00  ; 进料水平伺服上料位置设定按钮  HMI
MOVL(498) D416 D100  ; 进料水平伺服当前脉冲, 进料水平伺服上料位置脉冲
LD TR0
AND W100.01  ; 进料水平伺服左爪OK配对位置设定按钮  HMI
MOVL(498) D416 D102  ; 进料水平伺服当前脉冲, 进料水平伺服左爪OK配对位参数设定 (M)
LD TR0
AND W100.02  ; 进料水平伺服右爪OK配对位置设定按钮  HMI
MOVL(498) D416 D104  ; 进料水平伺服当前脉冲, 进料水平伺服右爪OK配对位参数设定 (M)
LD TR0
AND W100.03  ; 进料水平伺服左爪缓存位置设定按钮  HMI
MOVL(498) D416 D106  ; 进料水平伺服当前脉冲, 进料水平伺服右爪OK配对位参数设定 (M)
LD TR0
AND W100.04  ; 进料水平伺服右爪缓存位置设定按钮  HMI
MOVL(498) D416 D108  ; 进料水平伺服当前脉冲, 进料水平伺服右爪缓存位参数设定 (M)
LD TR0
AND W100.05  ; 进料水平伺服缓存位置设定按钮  HMI
MOVL(498) D416 D110  ; 进料水平伺服当前脉冲, 进料水平伺服左爪缓存位参数设定 (M)
LD TR0
AND W100.09  ; 进料水平伺服放料位置设定按钮  HMI
MOVL(498) D416 D118  ; 进料水平伺服当前脉冲, 进料水平伺服缓存位参数设定 (M)

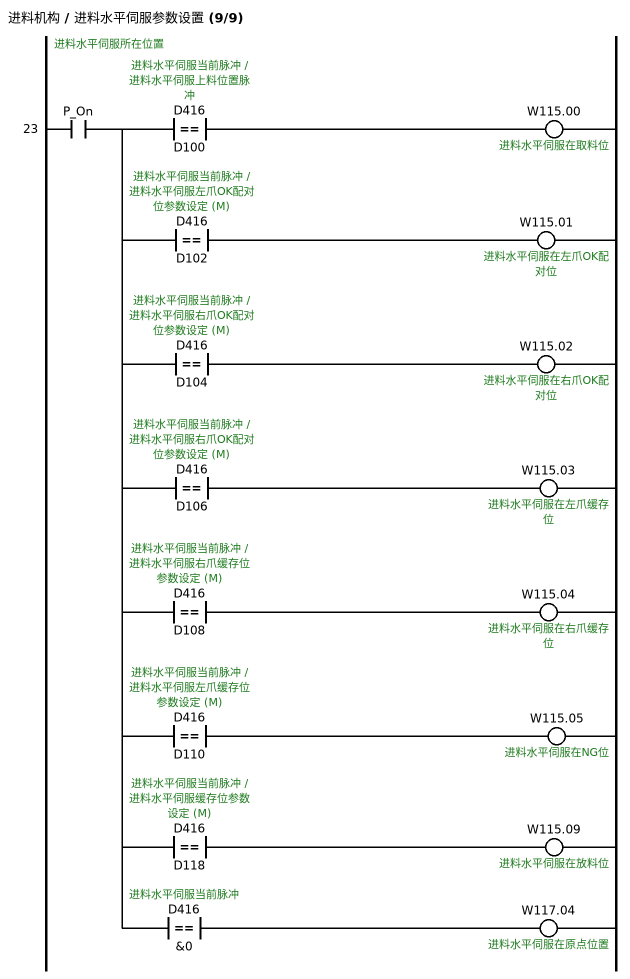
; rung 23: 进料水平伺服所在位置
LD P_On
OUT TR0
AND=SL(303) D416 D100  ; 进料水平伺服当前脉冲, 进料水平伺服上料位置脉冲
OUT W115.00  ; 进料水平伺服在取料位
LD TR0
AND=SL(303) D416 D102  ; 进料水平伺服当前脉冲, 进料水平伺服左爪OK配对位参数设定 (M)
OUT W115.01  ; 进料水平伺服在左爪OK配对位
LD TR0
AND=SL(303) D416 D104  ; 进料水平伺服当前脉冲, 进料水平伺服右爪OK配对位参数设定 (M)
OUT W115.02  ; 进料水平伺服在右爪OK配对位
LD TR0
AND=SL(303) D416 D106  ; 进料水平伺服当前脉冲, 进料水平伺服右爪OK配对位参数设定 (M)
OUT W115.03  ; 进料水平伺服在左爪缓存位
LD TR0
AND=SL(303) D416 D108  ; 进料水平伺服当前脉冲, 进料水平伺服右爪缓存位参数设定 (M)
OUT W115.04  ; 进料水平伺服在右爪缓存位
LD TR0
AND=SL(303) D416 D110  ; 进料水平伺服当前脉冲, 进料水平伺服左爪缓存位参数设定 (M)
OUT W115.05  ; 进料水平伺服在NG位
LD TR0
AND=SL(303) D416 D118  ; 进料水平伺服当前脉冲, 进料水平伺服缓存位参数设定 (M)
OUT W115.09  ; 进料水平伺服在放料位
LD TR0
AND=SL(303) D416 &0  ; 进料水平伺服当前脉冲
OUT W117.04  ; 进料水平伺服在原点位置

### Section 进料升降伺服参数设置

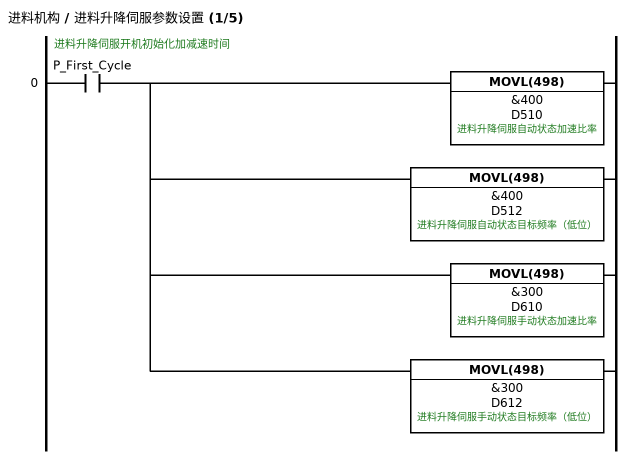
; rung 0: 进料升降伺服开机初始化加减速时间
LD P_First_Cycle
MOVL(498) &400 D510  ; 进料升降伺服自动状态加速比率
MOVL(498) &400 D512  ; 进料升降伺服自动状态目标频率（低位）
MOVL(498) &300 D610  ; 进料升降伺服手动状态加速比率
MOVL(498) &300 D612  ; 进料升降伺服手动状态目标频率（低位）

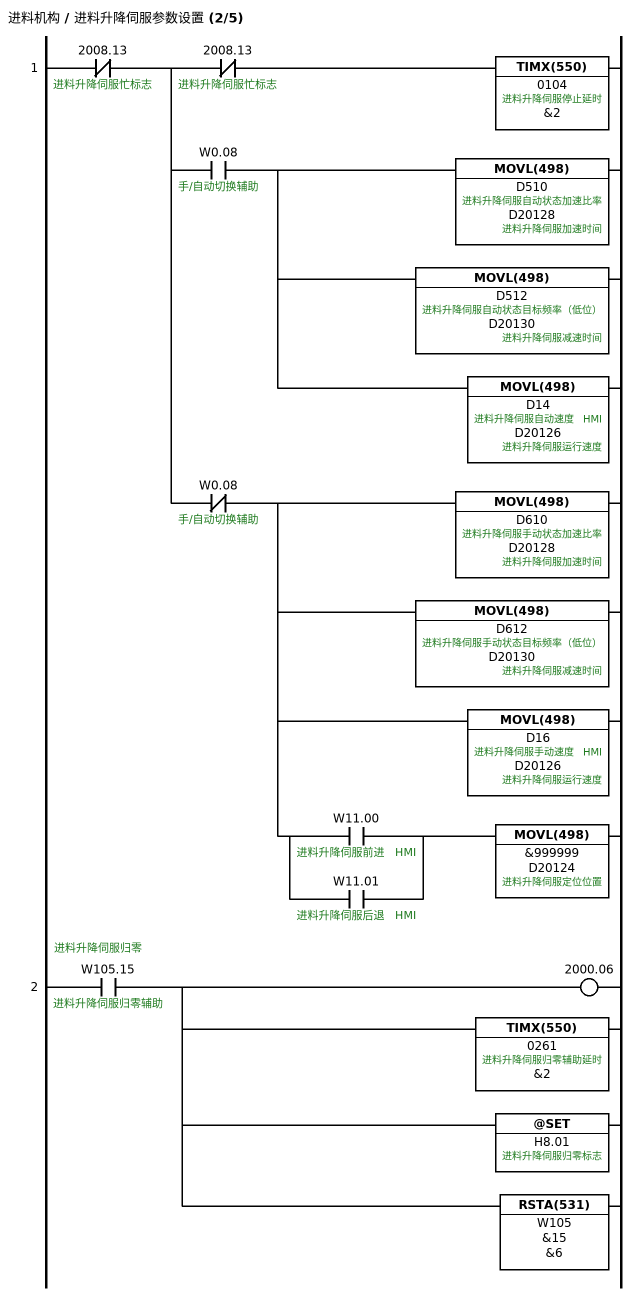
; rung 1
LDNOT 2008.13  ; 进料升降伺服忙标志
OUT TR0
ANDNOT 2008.13  ; 进料升降伺服忙标志
TIMX(550) 0104 &2  ; 进料升降伺服停止延时
LD TR0
AND W0.08  ; 手/自动切换辅助
MOVL(498) D510 D20128  ; 进料升降伺服自动状态加速比率, 进料升降伺服加速时间
MOVL(498) D512 D20130  ; 进料升降伺服自动状态目标频率（低位）, 进料升降伺服减速时间
MOVL(498) D14 D20126  ; 进料升降伺服自动速度   HMI, 进料升降伺服运行速度
LD TR0
ANDNOT W0.08  ; 手/自动切换辅助
MOVL(498) D610 D20128  ; 进料升降伺服手动状态加速比率, 进料升降伺服加速时间
MOVL(498) D612 D20130  ; 进料升降伺服手动状态目标频率（低位）, 进料升降伺服减速时间
MOVL(498) D16 D20126  ; 进料升降伺服手动速度   HMI, 进料升降伺服运行速度
LD W11.00  ; 进料升降伺服前进   HMI
OR W11.01  ; 进料升降伺服后退   HMI
ANDLD
MOVL(498) &999999 D20124  ; 进料升降伺服定位位置
; rung 2: 进料升降伺服归零
LD W105.15  ; 进料升降伺服归零辅助
OUT 2000.06
TIMX(550) 0261 &2  ; 进料升降伺服归零辅助延时
@SET H8.01  ; 进料升降伺服归零标志
RSTA(531) W105 &15 &6

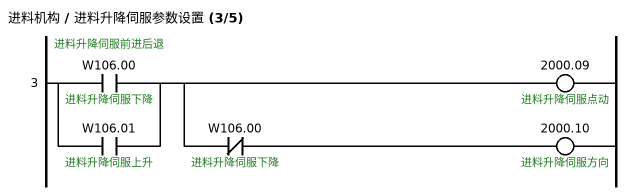
; rung 3: 进料升降伺服前进后退
LD W106.00  ; 进料升降伺服下降
OR W106.01  ; 进料升降伺服上升
OUT 2000.09  ; 进料升降伺服点动
ANDNOT W106.00  ; 进料升降伺服下降
OUT 2000.10  ; 进料升降伺服方向

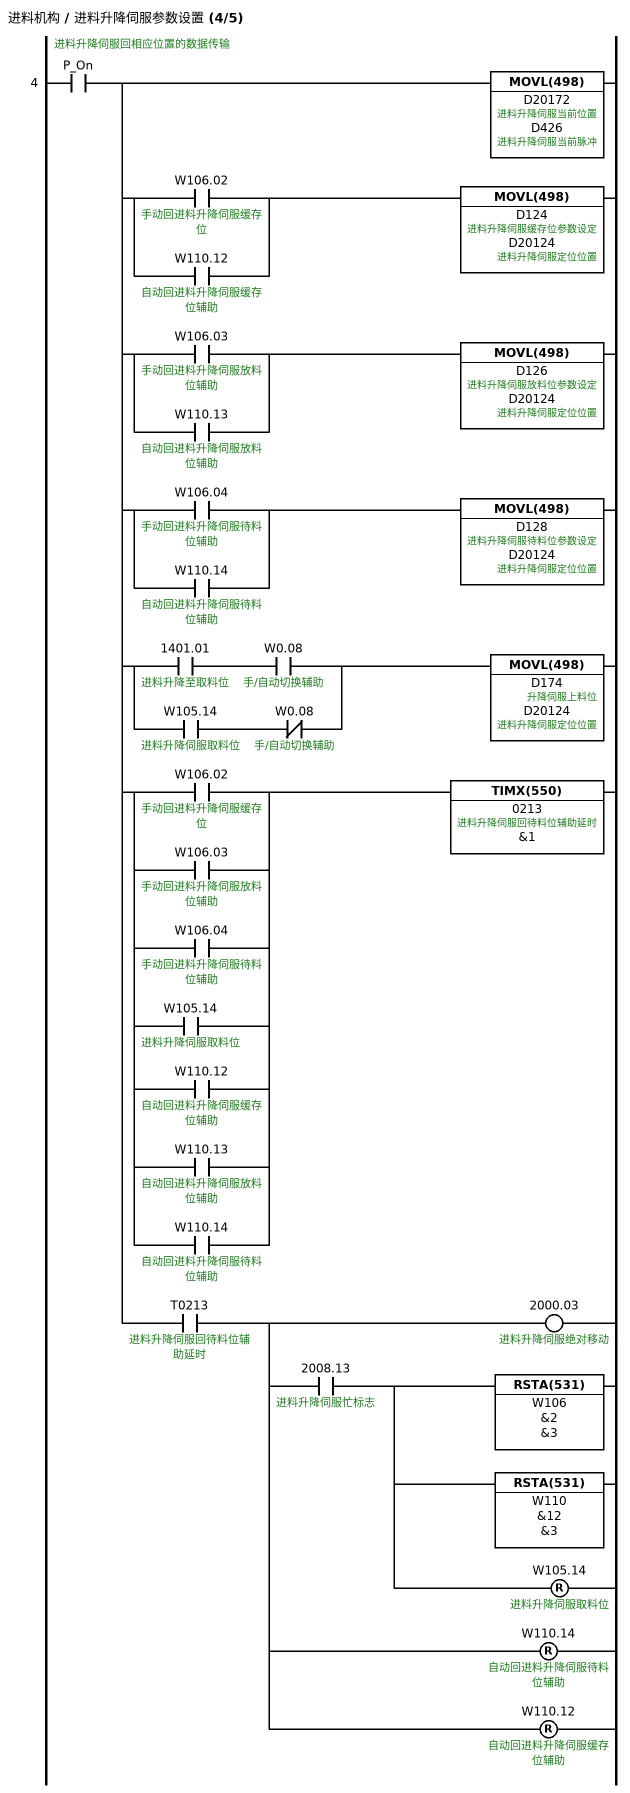
; rung 4: 进料升降伺服回相应位置的数据传输
LD P_On
OUT TR0
MOVL(498) D20172 D426  ; 进料升降伺服当前位置, 进料升降伺服当前脉冲
LD W106.02  ; 手动回进料升降伺服缓存位
OR W110.12  ; 自动回进料升降伺服缓存位辅助
ANDLD
MOVL(498) D124 D20124  ; 进料升降伺服缓存位参数设定, 进料升降伺服定位位置
LD TR0
LD W106.03  ; 手动回进料升降伺服放料位辅助
OR W110.13  ; 自动回进料升降伺服放料位辅助
ANDLD
MOVL(498) D126 D20124  ; 进料升降伺服放料位参数设定, 进料升降伺服定位位置
LD TR0
LD W106.04  ; 手动回进料升降伺服待料位辅助
OR W110.14  ; 自动回进料升降伺服待料位辅助
ANDLD
MOVL(498) D128 D20124  ; 进料升降伺服待料位参数设定, 进料升降伺服定位位置
LD TR0
LD 1401.01  ; 进料升降至取料位
AND W0.08  ; 手/自动切换辅助
LD W105.14  ; 进料升降伺服取料位
ANDNOT W0.08  ; 手/自动切换辅助
ORLD
ANDLD
MOVL(498) D174 D20124  ; 升降伺服上料位, 进料升降伺服定位位置
LD TR0
LD W106.02  ; 手动回进料升降伺服缓存位
OR W106.03  ; 手动回进料升降伺服放料位辅助
OR W106.04  ; 手动回进料升降伺服待料位辅助
OR W105.14  ; 进料升降伺服取料位
OR W110.12  ; 自动回进料升降伺服缓存位辅助
OR W110.13  ; 自动回进料升降伺服放料位辅助
OR W110.14  ; 自动回进料升降伺服待料位辅助
ANDLD
TIMX(550) 0213 &1  ; 进料升降伺服回待料位辅助延时
LD TR0
AND T0213  ; 进料升降伺服回待料位辅助延时
OUT TR0
OUT 2000.03  ; 进料升降伺服绝对移动
AND 2008.13  ; 进料升降伺服忙标志
RSTA(531) W106 &2 &3
RSTA(531) W110 &12 &3
RSET W105.14  ; 进料升降伺服取料位
LD TR0
RSET W110.14  ; 自动回进料升降伺服待料位辅助
RSET W110.12  ; 自动回进料升降伺服缓存位辅助

